// TIA Portal V18 export
FUNCTION_BLOCK "NG_BOXES"   // FB3, SCL
{ S7_Optimized_Access := 'TRUE' }
// stored: MemoryReserve 1000, SetENOAutomatically false
   VAR_INPUT
      in_Permission_to_Open : Bool;
   END_VAR
   VAR_OUTPUT
      out_Request_to_open : Bool;
   END_VAR
   VAR
      Box_Loading { S7_SetPoint := 'True'} : "FB_NG_Box_Control";
      Box_Unloading { S7_SetPoint := 'True'} : "FB_NG_Box_Control";
      TempSensors : Array[1..15] of Bool;
   END_VAR
BEGIN
   // ==========================================================================
   // BOX 1: LOADING – MACHINE LOADING SIDE                                   // EN: Loading side of machine (material IN)
   //                                                                          // CN: 机器上料侧（物料进入机器）
   //                                                                          // SK: Nakladacia / vstupná strana stroja
   // ==========================================================================
   #TempSensors[1] := "iE1-UnloadingShaftPressNG_1";   // EN: NG shaft press pos 1   // CN: 轴压装NG位置1   // SK: NG lis hriadeľa poz.1
   #TempSensors[2] := "iE1-UnloadingShaftPressNG_2";   // EN: NG shaft press pos 2   // CN: 轴压装NG位置2   // SK: NG lis hriadeľa poz.2
   #TempSensors[3] := "iE1-UnloadingShaftPressNG_3";   // EN: NG shaft press pos 3   // CN: 轴压装NG位置3   // SK: NG lis hriadeľa poz.3
   #TempSensors[4] := "iE1-UnloadingShaftPressNG_4";   // EN: NG shaft press pos 4   // CN: 轴压装NG位置4   // SK: NG lis hriadeľa poz.4
   #TempSensors[5] := "iE1-UnloadingShaftPressNG_5";   // EN: NG shaft press pos 5   // CN: 轴压装NG位置5   // SK: NG lis hriadeľa poz.5
   #TempSensors[6] := "iE1-UnloadingShaftScanNG_1";    // EN: NG shaft scan pos 1    // CN: 轴扫描NG位置1   // SK: NG sken hriadeľa 1
   #TempSensors[7] := "iE1-UnloadingShaftScanNG_2";    // EN: NG shaft scan pos 2    // CN: 轴扫描NG位置2   // SK: NG sken hriadeľa 2
   #TempSensors[8] := "iE1-UnloadingShaftScanNG_3";    // EN: NG shaft scan pos 3    // CN: 轴扫描NG位置3   // SK: NG sken hriadeľa 3
   #TempSensors[9] := "iE1-UnloadingShaftScanNG_4";    // EN: NG shaft scan pos 4    // CN: 轴扫描NG位置4   // SK: NG sken hriadeľa 4
   #TempSensors[10] := "iE1-UnloadingShaftScanNG_5";    // EN: NG shaft scan pos 5    // CN: 轴扫描NG位置5   // SK: NG sken hriadeľa 5
   #TempSensors[11] := "iE1-UnloadingRingScanNG_1";     // EN: NG ring scan pos 1     // CN: 环扫描NG位置1   // SK: NG sken krúžku 1
   #TempSensors[12] := "iE1-UnloadingRingScanNG_2";     // EN: NG ring scan pos 2     // CN: 环扫描NG位置2   // SK: NG sken krúžku 2
   #TempSensors[13] := "iE1-UnloadingRingScanNG_3";     // EN: NG ring scan pos 3     // CN: 环扫描NG位置3   // SK: NG sken krúžku 3
   #TempSensors[14] := "iE1-UnloadingRingScanNG_4";     // EN: NG ring scan pos 4     // CN: 环扫描NG位置4   // SK: NG sken krúžku 4
   #TempSensors[15] := "iE1-UnloadingRingScanNG_5";     // EN: NG ring scan pos 5     // CN: 环扫描NG位置5   // SK: NG sken krúžku 5

   #Box_Loading(
                Button        := "iNG_Button1",                     // EN: Operator button (loading side)   // CN: 上料侧操作按钮   // SK: Tlačidlo obsluhy – loading
                MagnetSensor  := "iE-NG-01Detection",               // EN: Door closed sensor                // CN: 门关闭传感器     // SK: Snímač zatvorenia dverí
                LockedFB      := NOT "iE-NG-01 Safety Gate_UnLock", // EN: Lock feedback (locked)             // CN: 锁定反馈         // SK: Spätná väzba – zamknuté
                UnlockedFB    := "iE-NG-01 Safety Gate_UnLock",     // EN: Lock feedback (unlocked)           // CN: 解锁反馈         // SK: Spätná väzba – odomknuté
                AtSafePoint   := #in_Permission_to_Open,            // EN: Sequence at safe point (Step 111)  // CN: 序列在安全步骤   // SK: Sekvencia v bezpečnom kroku
                Sensors       := #TempSensors,
                UnlockCmd     => "ST10_NGGate1_DB"."sSafetyGate UnlockRequest", // EN: Unlock command // CN: 解锁命令 // SK: Príkaz na odomknutie
                LockCmd       => "ST10_NGGate1_DB"."sSafetyGate LockRequest",   // EN: Lock command   // CN: 上锁命令 // SK: Príkaz na zamknutie
                CylinderOpen  => "oE-NG-01NGLocationCylinderToHP",   // EN: Cylinder open (home)  // CN: 气缸打开 // SK: Otvoriť valec
                CylinderClose => "oE-NG-01NGLocationCylinderToWP",   // EN: Cylinder close (work) // CN: 气缸关闭 // SK: Zavrieť valec
                ButtonLight => "oNG_Button1"   ,                    // E,N: Button lamp           // CN: 按钮灯   // SK: Svetlo tlačidla
                Ready_1 => "AutoProcessControl".NG_1.Robot1PutPrimit_1   ,         // Status pro robota: Řada 1 (1-5) má místo // 机器人状态：第1排（1-5）有空位
                Ready_2 => "AutoProcessControl".NG_1.Robot1PutPrimit_2,
                Ready_3 => "AutoProcessControl".NG_1.Robot1PutPrimit_3

   );

   // ==========================================================================
   // BOX 2: UNLOADING – MACHINE UNLOADING SIDE                                // EN: Unloading side of machine (material OUT)
   //                                                                          // CN: 机器下料侧（物料离开机器）
   //                                                                          // SK: Vykladacia / výstupná strana stroja
   // ==========================================================================
   #TempSensors[1] := "iE2-UnloadingPressNG_1";          // EN: NG press pos 1   // CN: 压装NG位置1   // SK: NG lis poz.1
   #TempSensors[2] := "iE2-UnloadingPressNG_2";          // EN: NG press pos 2   // CN: 压装NG位置2   // SK: NG lis poz.2
   #TempSensors[3] := "iE2-UnloadingPressNG_3";          // EN: NG press pos 3   // CN: 压装NG位置3   // SK: NG lis poz.3
   #TempSensors[4] := "iE2-UnloadingPressNG_4";          // EN: NG press pos 4   // CN: 压装NG位置4   // SK: NG lis poz.4
   #TempSensors[5] := "iE2-UnloadingPressNG_5";          // EN: NG press pos 5   // CN: 压装NG位置5   // SK: NG lis poz.5
   #TempSensors[6] := "iE2-UnloadingMagentScanNG_1";     // EN: NG magnet scan 1 // CN: 磁体扫描NG1   // SK: NG magnet sken 1
   #TempSensors[7] := "iE2-UnloadingMagentScanNG_2";     // EN: NG magnet scan 2 // CN: 磁体扫描NG2   // SK: NG magnet sken 2
   #TempSensors[8] := "iE2-UnloadingMagentScanNG_3";     // EN: NG magnet scan 3 // CN: 磁体扫描NG3   // SK: NG magnet sken 3
   #TempSensors[9] := "iE2-UnloadingMagentScanNG_4";     // EN: NG magnet scan 4 // CN: 磁体扫描NG4   // SK: NG magnet sken 4
   #TempSensors[10] := "iE2-UnloadingMagentScanNG_5";     // EN: NG magnet scan 5 // CN: 磁体扫描NG5   // SK: NG magnet sken 5
   #TempSensors[11] := "iE2-UnloadingRingScanNG_1";       // EN: NG ring scan 1   // CN: 环扫描NG1     // SK: NG sken krúžku 1
   #TempSensors[12] := "iE2-UnloadingRingScanNG_2";       // EN: NG ring scan 2   // CN: 环扫描NG2     // SK: NG sken krúžku 2
   #TempSensors[13] := "iE2-UnloadingRingScanNG_3";       // EN: NG ring scan 3   // CN: 环扫描NG3     // SK: NG sken krúžku 3
   #TempSensors[14] := "iE2-UnloadingRingScanNG_4";       // EN: NG ring scan 4   // CN: 环扫描NG4     // SK: NG sken krúžku 4
   #TempSensors[15] := "iE2-UnloadingRingScanNG_5";       // EN: NG ring scan 5   // CN: 环扫描NG5     // SK: NG sken krúžku 5

   #Box_Unloading(
                  Button        := "iNG_Button2",                     // EN: Operator button (unloading side) // CN: 下料侧操作按钮 // SK: Tlačidlo obsluhy – unloading
                  MagnetSensor  := "iE-NG-02Detection",               // EN: Door closed sensor               // CN: 门关闭传感器   // SK: Snímač zatvorenia dverí
                  LockedFB      := NOT "iE-NG-02 Safety Gate_UnLock", // EN: Lock feedback (locked)            // CN: 锁定反馈       // SK: Spätná väzba – zamknuté
                  UnlockedFB    := "iE-NG-02 Safety Gate_UnLock",     // EN: Lock feedback (unlocked)          // CN: 解锁反馈       // SK: Spätná väzba – odomknuté
                  AtSafePoint   := #in_Permission_to_Open,
                  Sensors       := #TempSensors,
                  UnlockCmd     => "ST10_NGGate2_DB"."sSafetyGate UnlockRequest",
                  LockCmd       => "ST10_NGGate2_DB"."sSafetyGate LockRequest",
                  CylinderOpen  => "oE-NG-02NGLocationCylinderToHP",
                  CylinderClose => "oE-NG-02NGLocationCylinderToWP",
                  ButtonLight   => "oNG_Button2",
                  Ready_1 => "AutoProcessControl".NG_2.Robot3PutPrimit_1   ,         // Status pro robota: Řada 1 (1-5) má místo // 机器人状态：第1排（1-5）有空位
                  Ready_2 => "AutoProcessControl".NG_2.Robot3PutPrimit_2,
                  Ready_3 => "AutoProcessControl".NG_2.Robot3PutPrimit_3
   );

   // EN: Request pause of main sequence if any side requests opening
   // CN: 任一侧请求开门时，请求暂停主序列
   // SK: Požiadavka na pauzu hlavnej sekvencie, ak ktorákoľvek strana žiada otvorenie
   #out_Request_to_open := #Box_Loading.PauseReq OR #Box_Unloading.PauseReq;
END_FUNCTION_BLOCK
